// TIA Portal project "APD Gateway Customer Library Source_V17" (V17)

(* hardware
DEVICE "S7-1200 station_1"  S7-1200 Station
   slot 0: "Rack_0"  S7-1200 Rack  Rack  V1.0
   slot 1: "customer"  CPU 1215C AC/DC/Rly  6ES7 215-1BG40-0XB0  V4.0
DEVICE "GSD device_1"  GSD.Device.PN
   slot 0: "Rack"  Rack  V1.0
   slot 1: "profinet_to_adp_gateway"  Profinet_to_ADP_Gateway  6ES7 215-1BG40-0XB0  V4.0
      slot 0: "Message"  Message
      slot 1: "Interface"  Interface
         slot 1: "Port 1"  Port 1
         slot 2: "Port 2"  Port 2
*)

// ===== PLC "customer"  CPU 1215C AC/DC/Rly =====

VAR_GLOBAL CONSTANT   // PLC tag table "ADP Gateway Constants"
   "FONT_NORMAL_5" : SInt := 1;
   "FONT_NORMAL_7" : SInt := 2;
   "FONT_NORMAL_9" : SInt := 3;
   "FONT_NORMAL_11" : SInt := 4;
   "FONT_NORMAL_14" : SInt := 5;
   "FONT_NORMAL_15" : SInt := 6;
   "FONT_NORMAL_16" : SInt := 7;
   "FONT_NORMAL_22" : SInt := 8;
   "FONT_NORMAL_24" : SInt := 9;
   "FONT_NORMAL_30" : SInt := 10;
   "FONT_NORMAL_32" : SInt := 11;
   "FONT_NORMAL_40" : SInt := 12;
   "FONT_BOLD_5" : SInt := 13;
   "FONT_BOLD_7" : SInt := 14;
   "FONT_BOLD_9" : SInt := 15;
   "FONT_BOLD_11" : SInt := 16;
   "FONT_BOLD_14" : SInt := 17;
   "FONT_BOLD_15" : SInt := 18;
   "FONT_BOLD_16" : SInt := 19;
   "FONT_BOLD_22" : SInt := 20;
   "FONT_BOLD_24" : SInt := 21;
   "FONT_BOLD_30" : SInt := 22;
   "FONT_BOLD_32" : SInt := 23;
   "FONT_BOLD_40" : SInt := 24;
   "SCROLL_FASTEST" : SInt := 1;
   "SCROLL_FAST" : SInt := 2;
   "SCROLL_NORMAL" : SInt := 3;
   "SCROLL_SLOW" : SInt := 4;
   "SCROLL_SLOWEST" : SInt := 5;
   "HORIZONTAL_LEFT" : SInt := 1;
   "HORIZONTAL_RIGHT" : SInt := 2;
   "HORIZONTAL_CENTER" : SInt := 3;
   "VERTICAL_BOTTOM" : SInt := 1;
   "VERTICAL_MIDDLE" : SInt := 2;
   "VERTICAL_TOP" : SInt := 3;
   "VERTICAL_FILL" : SInt := 4;
   "FOREGROUND_COLOR_BLACK" : SInt := 1;
   "FOREGROUND_COLOR_RED" : SInt := 2;
   "FOREGROUND_COLOR_GREEN" : SInt := 3;
   "FOREGROUND_COLOR_YELLOW" : SInt := 4;
   "FOREGROUND_COLOR_MIX_1" : SInt := 5;
   "FOREGROUND_COLOR_MIX_2" : SInt := 6;
   "FOREGROUND_COLOR_MIX_3" : SInt := 7;
   "FOREGROUND_COLOR_MIX_4" : SInt := 8;
   "FOREGROUND_COLOR_BLUE" : SInt := 9;
   "FOREGROUND_COLOR_WHITE" : SInt := 10;
   "BACKGROUND_COLOR_BLACK" : SInt := 1;
   "BACKGROUND_COLOR_RED" : SInt := 2;
   "BACKGROUND_COLOR_GREEN" : SInt := 3;
   "BACKGROUND_COLOR_YELLOW" : SInt := 4;
   "FLASH_ON" : SInt := 1;
   "FLASH_OFF" : SInt := 2;
END_VAR

// folder: ADP Gateway Interface Types

TYPE "ADP_Gateway_Interface.UDT"
   STRUCT
      hardware_address : DInt;
      line_formats : Array[0..4] of "ADP_Gateway_Interface.Line_Format.UDT";
      format_segments : Array[0..17] of "ADP_Gateway_Interface.Format_Segment.UDT";
   END_STRUCT;
END_TYPE

TYPE "ADP_Gateway_Interface.Line_Format.UDT"
   STRUCT
      font : SInt := 1;
      scroll_speed : SInt := 1;
      vertical_alignment : SInt := 1;
      horizontal_alignment : SInt := 1;
      hold : SInt := 5;
   END_STRUCT;
END_TYPE

TYPE "ADP_Gateway_Interface.Format_Segment.UDT"
   STRUCT
      foreground_color : SInt := 1;
      background_color : SInt := 1;
      flash : SInt := 1;
      line_number : SInt := -1;
      text : String[46];
   END_STRUCT;
END_TYPE

// folder: ADP Gateway Interface Blocks

DATA_BLOCK "ADP_Gateway_Interface_Data"   // DB1
{ S7_Optimized_Access := 'TRUE' }
VERSION : 0.1
BEGIN
END_DATA_BLOCK

// folder: (top level)

ORGANIZATION_BLOCK "Main"   // OB1, LAD, ProgramCycle
TITLE = "Main Program Sweep (Cycle)"
{ S7_Optimized_Access := 'TRUE' }
VERSION : 0.1
   VAR_INPUT
      Initial_Call : Bool;   // Initial call of this OB
      Remanence : Bool;   // =True, if remanent data are available
   END_VAR
BEGIN

REGION Network 1 (SCL)
   "ADP_Gateway_Interface_Data".hardware_address := 0;

   "ADP_Gateway_Interface_Data".line_formats[0].font := "FONT_BOLD_14";
   "ADP_Gateway_Interface_Data".line_formats[0].horizontal_alignment := "HORIZONTAL_LEFT";
   "ADP_Gateway_Interface_Data".line_formats[0].scroll_speed := "SCROLL_NORMAL";

   "ADP_Gateway_Interface_Data".format_segments[0].foreground_color := "FOREGROUND_COLOR_RED";
   "ADP_Gateway_Interface_Data".format_segments[0].flash := "FLASH_OFF";
END_REGION

REGION Network 2
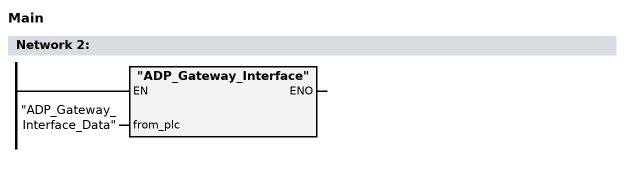
   RUNG wire#powerrail
      "ADP_Gateway_Interface"(from_plc := "ADP_Gateway_Interface_Data")
   END_RUNG
   // the same network as SCL:
   "ADP_Gateway_Interface"(from_plc := "ADP_Gateway_Interface_Data");
END_REGION
END_ORGANIZATION_BLOCK

// folder: ADP Gateway Interface Blocks

FUNCTION "ADP_Gateway_Interface" : Void   // FC1, SCL
TITLE = ADP Gateway Interface
{ S7_Optimized_Access := 'TRUE' }
AUTHOR : Machado
VERSION : 0.1
// for use with GSD file version xxxxx
   VAR_INPUT
      from_plc : "ADP_Gateway_Interface.UDT";
   END_VAR
   VAR_TEMP
      i : Int;
   END_VAR
   VAR CONSTANT
      LINE_COUNT : DInt := 4;   // 5 lines, 0 indexed
      FORMAT_SEGMENT_COUNT : DInt := 17;   // 18 format segments, 0 indexed
   END_VAR
BEGIN
   REGION LINE FORMATS
       FOR #i := 0 TO #LINE_COUNT DO
           "ADP_Gateway_Interface.Poke_Line_Formatting"(base_offset := 0,
                                                        from_plc := #from_plc.line_formats[#i],
                                                        line_number := #i);
       END_FOR;
   END_REGION


   REGION FORMAT SEGMENTS
       FOR #i := 0 TO #FORMAT_SEGMENT_COUNT DO
           "ADP_Gateway_Interface.Poke_Format_Segment"(base_offset := 50,
                                                       segment_number := #i,
                                                       format_segment := #from_plc.format_segments[#i]);
       END_FOR;
   END_REGION


   RETURN;
END_FUNCTION

FUNCTION "ADP_Gateway_Interface.Poke_Line_Formatting" : Void   // FC2, SCL
{ S7_Optimized_Access := 'TRUE' }
VERSION : 0.1
   VAR_INPUT
      base_offset : DInt;
      from_plc : "ADP_Gateway_Interface.Line_Format.UDT";
      line_number : Int;
   END_VAR
   VAR_TEMP
      offset : DInt;
   END_VAR
   VAR CONSTANT
      BYTES_PER_LINE : DInt := 5;
      OUTPUT_AREA : Byte := 16#82;
      NO_DB : DInt;
   END_VAR
BEGIN
   REGION BASE OFFSET
       #offset := #line_number * #BYTES_PER_LINE + #base_offset;
   END_REGION


   REGION FONT
       POKE(area := #OUTPUT_AREA,
            dbNumber := #NO_DB,
            byteOffset := #offset,
            value := SINT_TO_BYTE(#from_plc.font));
   END_REGION


   REGION SCROLL SPEED
       POKE(area := #OUTPUT_AREA,
            dbNumber := #NO_DB,
            byteOffset := #offset + 1,
            value := SINT_TO_BYTE(#from_plc.scroll_speed));
   END_REGION


   REGION VERTICAL ALIGNMENT
       POKE(area := #OUTPUT_AREA,
            dbNumber := #NO_DB,
            byteOffset := #offset + 2,
            value := SINT_TO_BYTE(#from_plc.vertical_alignment));
   END_REGION


   REGION HORIZONTAL ALIGNMENT
       POKE(area := #OUTPUT_AREA,
            dbNumber := #NO_DB,
            byteOffset := #offset + 3,
            value := SINT_TO_BYTE(#from_plc.horizontal_alignment));
   END_REGION


   REGION HOLD
       POKE(area := #OUTPUT_AREA,
            dbNumber := #NO_DB,
            byteOffset := #offset + 4,
            value := SINT_TO_BYTE(#from_plc.hold));
   END_REGION


   RETURN;
END_FUNCTION

FUNCTION "ADP_Gateway_Interface.Poke_Format_Segment" : Void   // FC3, SCL
{ S7_Optimized_Access := 'TRUE' }
VERSION : 0.1
   VAR_INPUT
      base_offset : DInt;
      segment_number : DInt;
      format_segment : "ADP_Gateway_Interface.Format_Segment.UDT";
   END_VAR
   VAR_TEMP
      i : DInt;
      offset : DInt;
   END_VAR
   VAR CONSTANT
      BYTES_PER_AREA : DInt := 50;
      BYTES_OF_TEXT : DInt := 49;
      OUTPUT_AREA : Byte := 16#82;
      NO_DB : DInt;
   END_VAR
BEGIN
   REGION BASE OFFSET
       #offset := #base_offset + #segment_number * #BYTES_PER_AREA;
   END_REGION


   REGION FOREGROUND
       POKE(area := #OUTPUT_AREA,
            dbNumber := #NO_DB,
            byteOffset := #offset,
            value := SINT_TO_BYTE(#format_segment.foreground_color));
   END_REGION


   REGION BACKGROUND
       POKE(area := #OUTPUT_AREA,
            dbNumber := #NO_DB,
            byteOffset := #offset + 1,
            value := SINT_TO_BYTE(#format_segment.background_color));
   END_REGION


   REGION FLASH
       POKE(area := #OUTPUT_AREA,
            dbNumber := #NO_DB,
            byteOffset := #offset + 2,
            value := SINT_TO_BYTE(#format_segment.flash));
   END_REGION


   REGION LINE NUMBER
       POKE(area := #OUTPUT_AREA,
            dbNumber := #NO_DB,
            byteOffset := #offset + 3,
            value := SINT_TO_BYTE(#format_segment.line_number));
   END_REGION


   REGION TEXT
       FOR #i := 0 TO #BYTES_OF_TEXT DO
           POKE(area := #OUTPUT_AREA,
                dbNumber := #NO_DB,
                byteOffset := #offset + #i + 4,
                value := CHAR_TO_BYTE(#format_segment.text[#i]));
       END_FOR;
   END_REGION
END_FUNCTION